Staubli VAL3: StackCount.dtx

mdesc mNomSpeed
num nNum = 88
string sString
